(* Logix 5000 project; controller RA_Base vendor 1 type 14 code 94 rev 32.11; software revision 32.00 *)

TASK MainTask (continuous, watchdog 1000 ms) : MainProgram

MODULES
   Local : vendor 1 type 14 code 94 (ICP 0, rev 32.11)
      S4_IF8H : vendor 1 type 10 code 114 (ICP 4, rev 2.1, Input RPI 100 ms)
           Local:4:I.Ch0Data   // Feedback Posicion FV10
           Local:4:I.Ch1Data   // Feedback Posicion FV11
           Local:4:I.Ch2Data   // PT10 Presion 1 Tanque de Proceso
           Local:4:I.Ch3Data   // PT11 Presion 2 Tanque de Proceso
           Local:4:I.Ch4Data   // PT20 Presion Descarga de Bomba VFD10
           Local:4:I.Ch5Data   // TT10 Temperatura Tanque de Proceso
           Local:4:I.Ch6Data   // TT10 Temperatura Tanque de Agua Caliente
      S5_OF8H : vendor 1 type 10 code 115 (ICP 5, rev 2.1, Output RPI 25 ms)
      R0_S2_EN2T : 1756-EN2T (Ethernet 192.168.1.4, ICP 2, rev 10.1)
      EN2TR : vendor 1 type 12 code 200 (ICP 1, Ethernet 192.168.1.10, rev 10.1)
         POWERFLEX_525 : PowerFlex 525-EENET (Ethernet 192.168.1.15, rev 4.1, Output RPI 20 ms)
         FLEXIO : 1794-AENTR (Ethernet 192.168.1.12, rev 1.1, Output RPI 20 ms)
            S0_IB16 : 1794-IB16 (Flex 0, rev 1.1)
            S1_OB16 : vendor 1 type 7 code 35 (Flex 1, rev 1.1)
            S2_RIE8XOE4 : vendor 1 type 10 code 113 (Flex 2, rev 1.1, Output RPI 80 ms)
      PROSOFT_PROFIBUSDP : vendor 1 type 0 code 15 (ICP 3, rev 1.1, Output RPI 5 ms)
END_MODULES

TYPE Port_Name :
STRUCT
   LEN : DINT;
   DATA : SINT[8];
END_STRUCT
END_TYPE

TYPE STRING128 :
STRUCT
   LEN : DINT;
   DATA : SINT[128];
END_STRUCT
END_TYPE

TYPE STRING32 :
STRUCT
   LEN : DINT;
   DATA : SINT[32];
END_STRUCT
END_TYPE

TYPE STRING64 :
STRUCT
   LEN : DINT;
   DATA : SINT[64];
END_STRUCT
END_TYPE

TYPE STRING_12 :
STRUCT
   LEN : DINT;
   DATA : SINT[12];
END_STRUCT
END_TYPE

TYPE STRING_16 :
STRUCT
   LEN : DINT;
   DATA : SINT[16];
END_STRUCT
END_TYPE

TYPE STRING_20 :
STRUCT
   LEN : DINT;
   DATA : SINT[20];
END_STRUCT
END_TYPE

TYPE STRING_40 :
STRUCT
   LEN : DINT;
   DATA : SINT[40];
END_STRUCT
END_TYPE

TYPE STRING_8 :
STRUCT
   LEN : DINT;
   DATA : SINT[8];
END_STRUCT
END_TYPE

PROGRAM MainProgram   (* main routine MainRoutine *)
VAR
   APAGAR : BOOL;
   cierre : TIMER := (PRE := 1000);
   DESACTIVA : BOOL;
   DESACTIVA2 : BOOL;
   DV10 : ALIAS FOR FLEXIO:1:O.0;
   DV10_VER : ALIAS FOR FLEXIO:0:I.0;
   DV20 : ALIAS FOR FLEXIO:1:O.1;
   DV20_VER : ALIAS FOR FLEXIO:0:I.1;
   DV30 : ALIAS FOR FLEXIO:1:O.2;
   FV10 : ALIAS FOR Local:5:O.Ch1Data;
   FV10_VER : ALIAS FOR Local:4:I.Ch1Data;
   FV11 : ALIAS FOR Local:5:O.Ch0Data;
   FV11_VER : ALIAS FOR Local:4:I.Ch0Data;
   INICIA : BOOL;
   LAH : ALIAS FOR Local:4:I.Ch2Data;
   LAHH : ALIAS FOR FLEXIO:0:I.3;
   LALL : ALIAS FOR FLEXIO:0:I.4;
   S1 : BOOL;
   S2 : BOOL;
END_VAR

ROUTINE MainRoutine   (* ladder *)
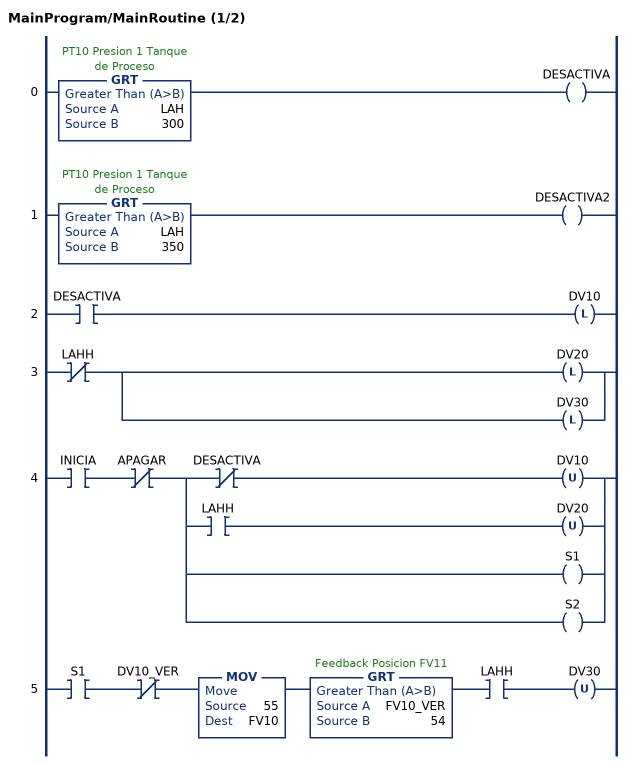
   0: GRT(LAH,300)OTE(DESACTIVA);
   1: GRT(LAH,350)OTE(DESACTIVA2);
   2: XIC(DESACTIVA)OTL(DV10);
   3: XIO(LAHH)[OTL(DV20) ,OTL(DV30) ];
   4: XIC(INICIA)XIO(APAGAR)[XIO(DESACTIVA) OTU(DV10) ,[XIC(LAHH) OTU(DV20) ,[OTE(S1) ,OTE(S2) ] ] ];
   5: XIC(S1)XIO(DV10_VER)MOV(55,FV10)GRT(FV10_VER,54)XIC(LAHH)OTU(DV30);
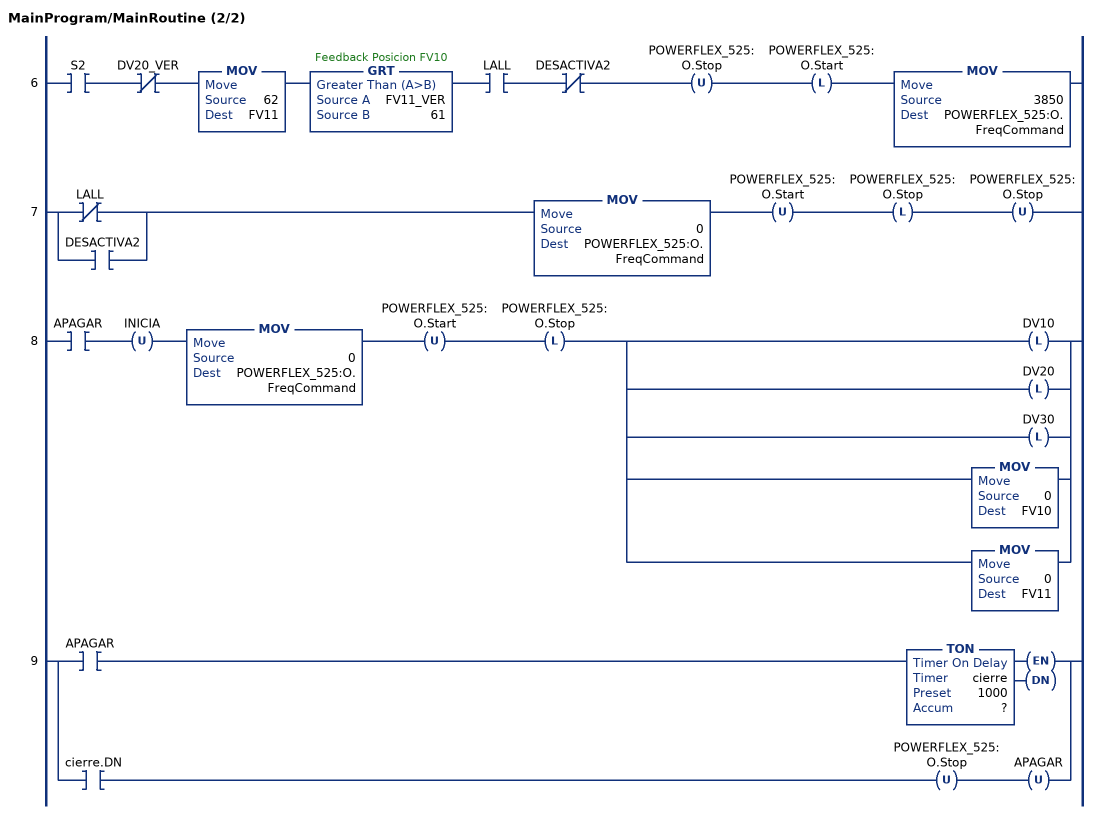
   6: XIC(S2)XIO(DV20_VER)MOV(62,FV11)GRT(FV11_VER,61)XIC(LALL)XIO(DESACTIVA2)OTU(POWERFLEX_525:O.Stop)OTL(POWERFLEX_525:O.Start)MOV(3850,POWERFLEX_525:O.FreqCommand);
   7: [XIO(LALL) ,XIC(DESACTIVA2) ]MOV(0,POWERFLEX_525:O.FreqCommand)OTU(POWERFLEX_525:O.Start)OTL(POWERFLEX_525:O.Stop)OTU(POWERFLEX_525:O.Stop);
   8: XIC(APAGAR)OTU(INICIA)MOV(0,POWERFLEX_525:O.FreqCommand)OTU(POWERFLEX_525:O.Start)OTL(POWERFLEX_525:O.Stop)[OTL(DV10) ,[OTL(DV20) ,[OTL(DV30) ,[MOV(0,FV10) ,MOV(0,FV11) ] ] ] ];
   9: [XIC(APAGAR) TON(cierre,?,?) ,XIC(cierre.DN) OTU(POWERFLEX_525:O.Stop) OTU(APAGAR) ];
END_ROUTINE
END_PROGRAM
